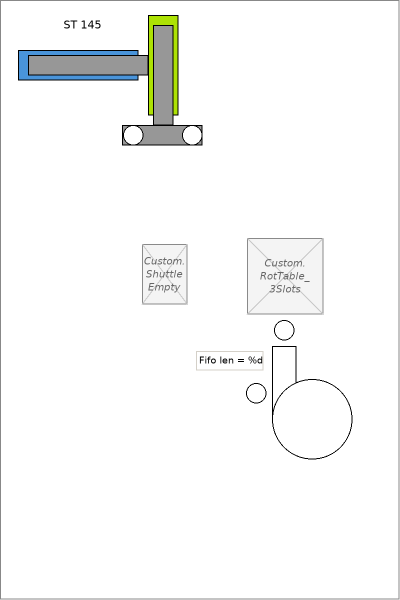
VISUALIZATION VISU_ST145  // 400x600
    Image (142,244 45x60), invisible if: NOT __ISVALIDREF(GVL._Process9._Mover), image: Custom.Shuttle Empty
    Image (247,238 76x76), image: Custom.RotTable_3Slots
        p2858320360: ST145_Axis.axis145_10W.axis.NcToPlc.ModuloActPos
    Rectangle (18,50 120x30)
    Rectangle (28,55 120x20)
        p3560616238: GVL._Process9.fb_Pnp.fb_simu_axis145_01Y.rOUT_PixActual
    Rectangle (148,15 30x100)
        p3560616238: GVL._Process9.fb_Pnp.fb_simu_axis145_01Y.rOUT_PixActual
    Rectangle (153,25 20x100)
        p2738717112: GVL._Process9.fb_Pnp.fb_simu_axis145_02Z.rOUT_PixActual
        p3560616238: GVL._Process9.fb_Pnp.fb_simu_axis145_01Y.rOUT_PixActual
    Rectangle (272,346 24x73)
    Ellipse (272,379 80x80), colour toggle: GVL._Process9.fb_Feeder.simu_feeder.xIN_Enable
    Ellipse (246,383 20x20), colour toggle: GVL._Process9.fb_Feeder.simu_feeder.xOUT_NewPiece
    Ellipse (274,320 20x20), colour toggle: NOT GVL._Process9.fb_Feeder.simu_fifo_feeder_to_rotTable.IsEmpty()
    Textfield (196,351 67x19), "Fifo len = %d", text variable: GVL._Process9.fb_Feeder.simu_fifo_feeder_to_rotTable.GetLen()
    Label (40,15 85x20), "ST 145"
    Rectangle (122,125 80x20)
        p2738717112: GVL._Process9.fb_Pnp.fb_simu_axis145_02Z.rOUT_PixActual
        p3560616238: GVL._Process9.fb_Pnp.fb_simu_axis145_01Y.rOUT_PixActual
    Ellipse (123,125 20x20), colour toggle: GVL._Process9.fb_Pnp.fb_vakumGriperLeft.xIN_AS
        p3560616238: GVL._Process9.fb_Pnp.fb_simu_axis145_01Y.rOUT_PixActual
        p2738717112: GVL._Process9.fb_Pnp.fb_simu_axis145_02Z.rOUT_PixActual
    Ellipse (182,125 20x20), colour toggle: GVL._Process9.fb_Pnp.fb_vakumGriperRight.xIN_AS
        p3560616238: GVL._Process9.fb_Pnp.fb_simu_axis145_01Y.rOUT_PixActual
        p2738717112: GVL._Process9.fb_Pnp.fb_simu_axis145_02Z.rOUT_PixActual
END_VISUALIZATION

(* stored: Version 1.1.0.1, ProductVersion 3.1.4024.6
   Visu VISU_ST145: Id {4e267c8e-f9b9-4178-93f1-39f373b002c6} *)
